% RSLogix 500 project projectplcwood.RSS, saved by version 8.30.00.16 %
PROJECT "UNTITLED"    % processor: MicroLogix 1000 %

PROGRAM FILES
  LAD 2 "MAIN_PROG"  9 rungs
  LAD 3 "USER_FAULT"  1 rungs
  LAD 4 "HSC_INT"  1 rungs
  LAD 5 "STI_INT"  1 rungs
  LAD 6, 7, 8, 9, 10, 11, 12, 13, 14, 15, 16: only END

DATA FILES
  O0 OUTPUT  1 elements
  I1 INPUT  2 elements
  S2 STATUS  33 elements
  B3 BINARY  32 elements
  T4 TIMER  40 elements
  C5 COUNTER  32 elements
  R6 CONTROL  16 elements
  N7 INTEGER  105 elements

LADDER 2 "MAIN_PROG"
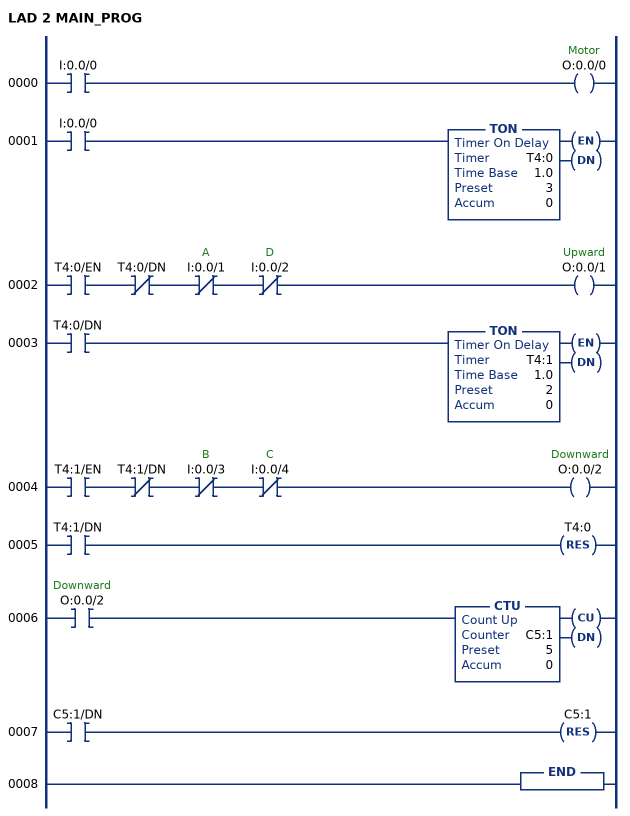
% Rung: 0 %
SOR XIC I:0.0/0 OTE O:0.0/0 EOR
%   O:0.0/0  "Motor" %
% Rung: 1 %
SOR XIC I:0.0/0 TON T4:0 1.0 3 0 EOR
% Rung: 2 %
SOR XIC T4:0/EN XIO T4:0/DN XIO I:0.0/1 XIO I:0.0/2 OTE O:0.0/1 EOR
%   I:0.0/1  "A" %
%   I:0.0/2  "D" %
%   O:0.0/1  "Upward" %
% Rung: 3 %
SOR XIC T4:0/DN TON T4:1 1.0 2 0 EOR
% Rung: 4 %
SOR XIC T4:1/EN XIO T4:1/DN XIO I:0.0/3 XIO I:0.0/4 OTE O:0.0/2 EOR
%   I:0.0/3  "B" %
%   I:0.0/4  "C" %
%   O:0.0/2  "Downward" %
% Rung: 5 %
SOR XIC T4:1/DN RES T4:0 EOR
% Rung: 6 %
SOR XIC O:0.0/2 CTU C5:1 5 0 EOR
%   O:0.0/2  "Downward" %
% Rung: 7 %
SOR XIC C5:1/DN RES C5:1 EOR
% Rung: 8 %
SOR END EOR

DATA TABLE (non-zero values as saved)
DATA T4
% .PRE .ACC %
% T4:0 % 3 0
% T4:1 % 2 0
DATA C5
% .PRE .ACC %
% C5:1 % 5 0
